Omron CX-Programmer project NuevoProyecto (CX-Programmer 9.73)

# PLC Practica3Diposits: CJ2M CPU31
I/O table (CPU CJ2M-CPU31): rack 0 slot 11 CJ2M-EIP21

## Program NuevoPrograma1 (cyclic task 0)
Local symbols
Base_1s W0.01 BOOL
Bomba1 H1.01 BOOL
Bomba2 H1.02 BOOL
Bomba3 H1.03 BOOL
Bomba_X_Activa W0.02 BOOL
Desague_Permitido W0.03 BOOL
Electrovalvula H1.04 BOOL
Litros_Deposito D100 UINT_BCD
Marcha H0.00 BOOL
Motor H2.00 BOOL
Numero_Bomba_Activa D51 UINT_BCD
Paro H0.01 BOOL
Pulso1_s CHANNEL
Pulso_1s W0.10 BOOL
Reset_Tempos H0.07 BOOL
Sistema_Actiu W0.00 BOOL
TickEnable W0.11 BOOL
TiempoBomba1 D1 UINT_BCD
TiempoBomba2 D2 UINT_BCD
TiempoBomba3 D3 UINT_BCD
TiempoCambio D53 UINT_BCD
Valor_Minimo D50 UINT_BCD
segundos_de_ciclo D52 UINT_BCD

### Section Sección1

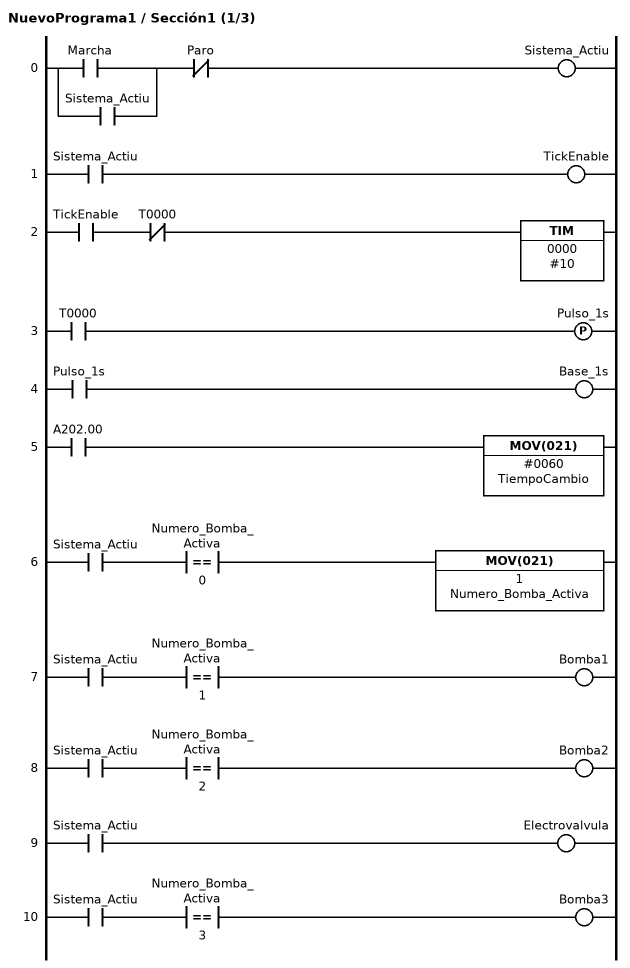
; rung 0
LD Marcha
OR Sistema_Actiu
ANDNOT Paro
OUT Sistema_Actiu
; rung 1
LD Sistema_Actiu
OUT TickEnable
; rung 2
LD TickEnable
ANDNOT T0000
TIM 0000 #10
; rung 3
LD T0000
DIFU(013) Pulso_1s
; rung 4
LD Pulso_1s
OUT Base_1s
; rung 5
LD A202.00
MOV(021) #0060 TiempoCambio
; rung 6
LD Sistema_Actiu
AND=(300) Numero_Bomba_Activa 0
MOV(021) 1 Numero_Bomba_Activa
; rung 7
LD Sistema_Actiu
AND=(300) Numero_Bomba_Activa 1
OUT Bomba1
; rung 8
LD Sistema_Actiu
AND=(300) Numero_Bomba_Activa 2
OUT Bomba2
; rung 9
LD Sistema_Actiu
OUT Electrovalvula
; rung 10
LD Sistema_Actiu
AND=(300) Numero_Bomba_Activa 3
OUT Bomba3

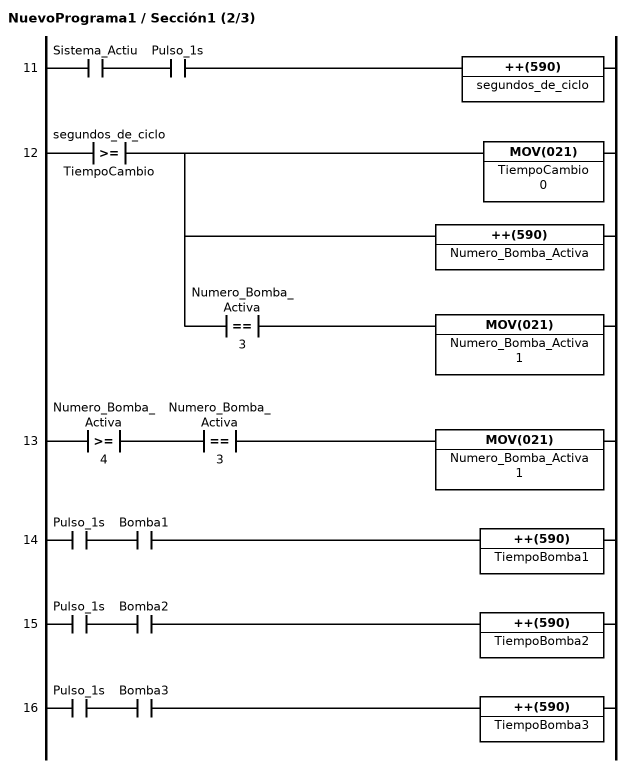
; rung 11
LD Sistema_Actiu
AND Pulso_1s
++(590) segundos_de_ciclo
; rung 12
LD>=(325) segundos_de_ciclo TiempoCambio
MOV(021) TiempoCambio 0
++(590) Numero_Bomba_Activa
AND=(300) Numero_Bomba_Activa 3
MOV(021) Numero_Bomba_Activa 1
; rung 13
LD>=(325) Numero_Bomba_Activa 4
AND=(300) Numero_Bomba_Activa 3
MOV(021) Numero_Bomba_Activa 1
; rung 14
LD Pulso_1s
AND Bomba1
++(590) TiempoBomba1
; rung 15
LD Pulso_1s
AND Bomba2
++(590) TiempoBomba2
; rung 16
LD Pulso_1s
AND Bomba3
++(590) TiempoBomba3

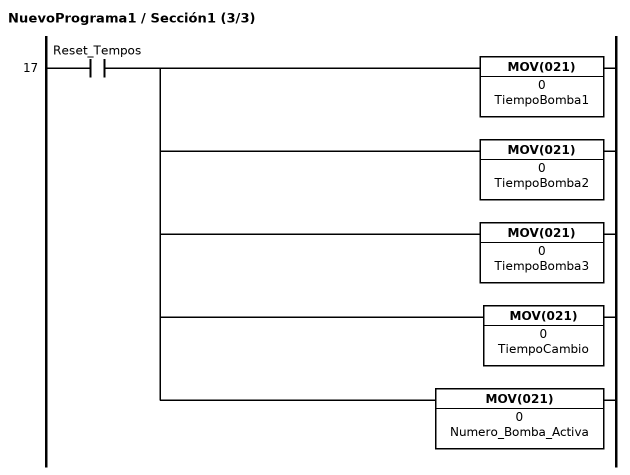
; rung 17
LD Reset_Tempos
MOV(021) 0 TiempoBomba1
MOV(021) 0 TiempoBomba2
MOV(021) 0 TiempoBomba3
MOV(021) 0 TiempoCambio
MOV(021) 0 Numero_Bomba_Activa

### Section END
; rung 0
END(001)